PROGRAM valve_manager
VAR
	//Digital valve
	nv_3110_b : valve_digital;
	nv_3210_b : valve_digital;
	nv_3310_b : valve_digital;
	nv_3135_b : valve_digital;
	nv_3235_b : valve_digital;
	nv_3335_b : valve_digital;
	nv_3372_b : valve_digital;
	nv_3162_b : valve_digital;
	
	// Analog Valve Function Block
	av_3148_b : valve_analog;
	av_3248_b : valve_analog;
	av_3348_b : valve_analog;


	//Repeat for each valve?
	u_3112_b_open_request: BOOL;
	u_3112_b_idle_request: BOOL;
	u_3112_b_cip_request: BOOL;
	u_3112_b_manual_request: BOOL;
	u_3112_b_stop_request: BOOL;
	u_3112_b_intlk: BOOL;
	gen_alm_active: BOOL;
	ed_routine_idle: BOOL;
	ed_routine_cip: BOOL;
	ed_routine_manual: BOOL;
	ed_routine_maint: BOOL;
	nv_3110_b_idle_request: BOOL;
	nv_3110_b_cip_request: BOOL;
	nv_3110_b_manual_request: BOOL;
	nv_3110_b_intlk: BOOL;
	nv_3110_b_stop_request: BOOL;
	nv_3110_b_open_request: BOOL;
	nv_3210_b_open_request: BOOL;
	nv_3310_b_open_request: BOOL;
	nv_3135_b_open_request: BOOL;
	nv_3235_b_open_request: BOOL;
	nv_3335_b_open_request: BOOL;
	nv_3372_b_open_request: BOOL;
	nv_3210_b_idle_request: BOOL;
	nv_3210_b_cip_request: BOOL;
	nv_3210_b_manual_request: BOOL;
	nv_3210_b_stop_request: BOOL;
	nv_3210_b_intlk: BOOL;
	
	nv_3310_b_idle_request: BOOL;
	nv_3310_b_cip_request: BOOL;
	nv_3310_b_manual_request: BOOL;
	nv_3310_b_stop_request: BOOL;
	nv_3310_b_intlk: BOOL;
	
	nv_3135_b_idle_request: BOOL;
	nv_3135_b_cip_request: BOOL;
	nv_3135_b_manual_request: BOOL;
	nv_3135_b_stop_request: BOOL;
	nv_3135_b_intlk: BOOL;
	
	nv_3235_b_idle_request: BOOL;
	nv_3235_b_cip_request: BOOL;
	nv_3235_b_manual_request: BOOL;
	nv_3235_b_stop_request: BOOL;
	nv_3235_b_intlk: BOOL;
	
	nv_3335_b_idle_request: BOOL;
	nv_3335_b_cip_request: BOOL;
	nv_3335_b_manual_request: BOOL;
	nv_3335_b_stop_request: BOOL;
	nv_3335_b_intlk: BOOL;
	
	nv_3372_b_idle_request: BOOL;
	nv_3372_b_cip_request: BOOL;
	nv_3372_b_manual_request: BOOL;
	nv_3372_b_stop_request: BOOL;
	nv_3372_b_intlk: BOOL;
	
	nv_3162_b_idle_request: BOOL;
	nv_3162_b_cip_request: BOOL;
	nv_3162_b_manual_request: BOOL;
	nv_3162_b_stop_request: BOOL;
	nv_3162_b_intlk: BOOL;
	nv_3162_b_open_request: BOOL;
	
	av_3148_b_idle_request: BOOL;
	av_3148_b_cip_request: BOOL;
	av_3148_b_idle_position_request: REAL;
	av_3148_b_position_request: REAL;
	av_3148_b_cip_position_request: REAL;
	av_3148_b_manual_position_request: REAL;
	av_3148_b_manual_request: BOOL;
	av_3148_b_maint_request: BOOL;
	av_3148_b_maint_position_request: REAL;
	av_3148_b_intlk: BOOL;
	av_3148_b_stop_request: BOOL;
	av_3148_b_open_request: BOOL;
	
	av_3248_b_idle_request: BOOL;
	av_3248_b_cip_request: BOOL;
	av_3248_b_idle_position_request: REAL;
	av_3248_b_position_request: REAL;
	av_3248_b_cip_position_request: REAL;
	av_3248_b_manual_position_request: REAL;
	av_3248_b_manual_request: BOOL;
	av_3248_b_maint_request: BOOL;
	av_3248_b_maint_position_request: REAL;
	av_3248_b_intlk: BOOL;
	av_3248_b_stop_request: BOOL;
	av_3248_b_open_request: BOOL;
	
	av_3348_b_idle_request: BOOL;
	av_3348_b_cip_request: BOOL;
	av_3348_b_idle_position_request: REAL;
	av_3348_b_position_request: REAL;
	av_3348_b_cip_position_request: REAL;
	av_3348_b_manual_position_request: REAL;
	av_3348_b_manual_request: BOOL;
	av_3348_b_maint_request: BOOL;
	av_3348_b_maint_position_request: REAL;
	av_3348_b_intlk: BOOL;
	av_3348_b_stop_request: BOOL;
	av_3348_b_open_request: BOOL;
	
END_VAR
VAR // added by the converter: edge detectors and wires of the graphical bodies
    _w1, _w2, _w3, _w4, _w5, _w6, _w7, _w8, _w9, _w10, _w11, _w12, _w13, _w14, _w15 : BOOL;
END_VAR

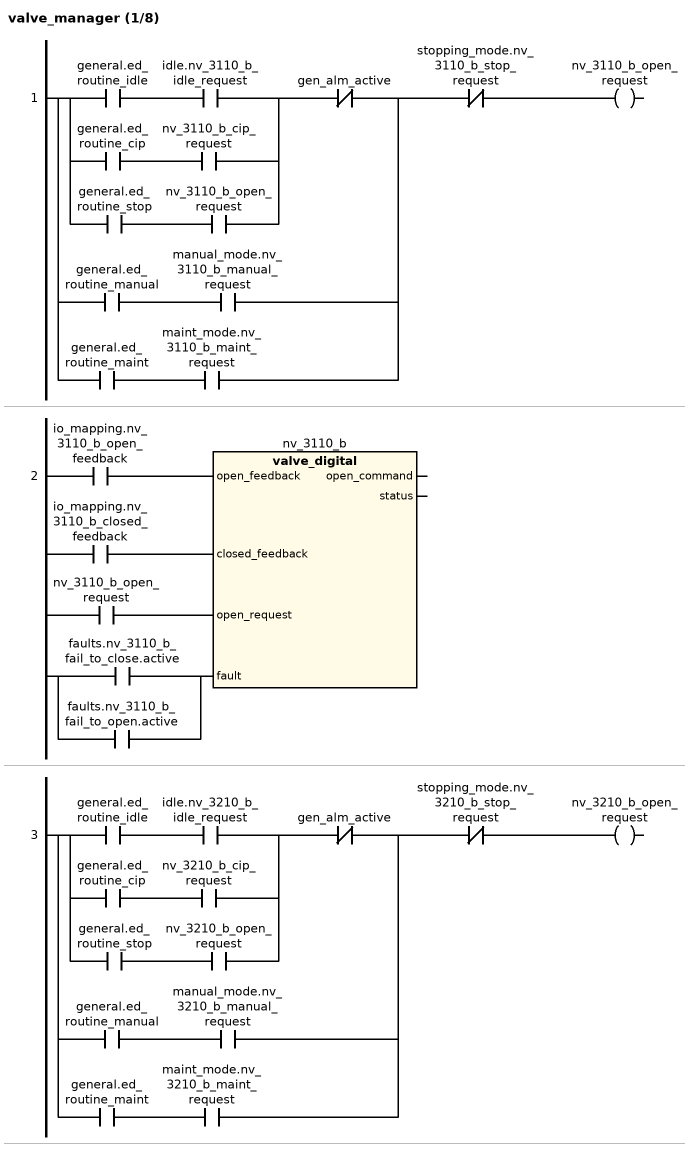
// NETWORK 1
nv_3110_b_open_request := ((general.ed_routine_idle AND idle.nv_3110_b_idle_request OR general.ed_routine_cip AND nv_3110_b_cip_request OR general.ed_routine_stop AND nv_3110_b_open_request) AND NOT gen_alm_active OR general.ed_routine_manual AND manual_mode.nv_3110_b_manual_request OR general.ed_routine_maint AND maint_mode.nv_3110_b_maint_request) AND NOT stopping_mode.nv_3110_b_stop_request;

// NETWORK 2
nv_3110_b(
    open_feedback := io_mapping.nv_3110_b_open_feedback,
    closed_feedback := io_mapping.nv_3110_b_closed_feedback,
    open_request := nv_3110_b_open_request,
    fault := faults.nv_3110_b_fail_to_close.active OR faults.nv_3110_b_fail_to_open.active); // valve_digital

// NETWORK 3
nv_3210_b_open_request := ((general.ed_routine_idle AND idle.nv_3210_b_idle_request OR general.ed_routine_cip AND nv_3210_b_cip_request OR general.ed_routine_stop AND nv_3210_b_open_request) AND NOT gen_alm_active OR general.ed_routine_manual AND manual_mode.nv_3210_b_manual_request OR general.ed_routine_maint AND maint_mode.nv_3210_b_maint_request) AND NOT stopping_mode.nv_3210_b_stop_request;

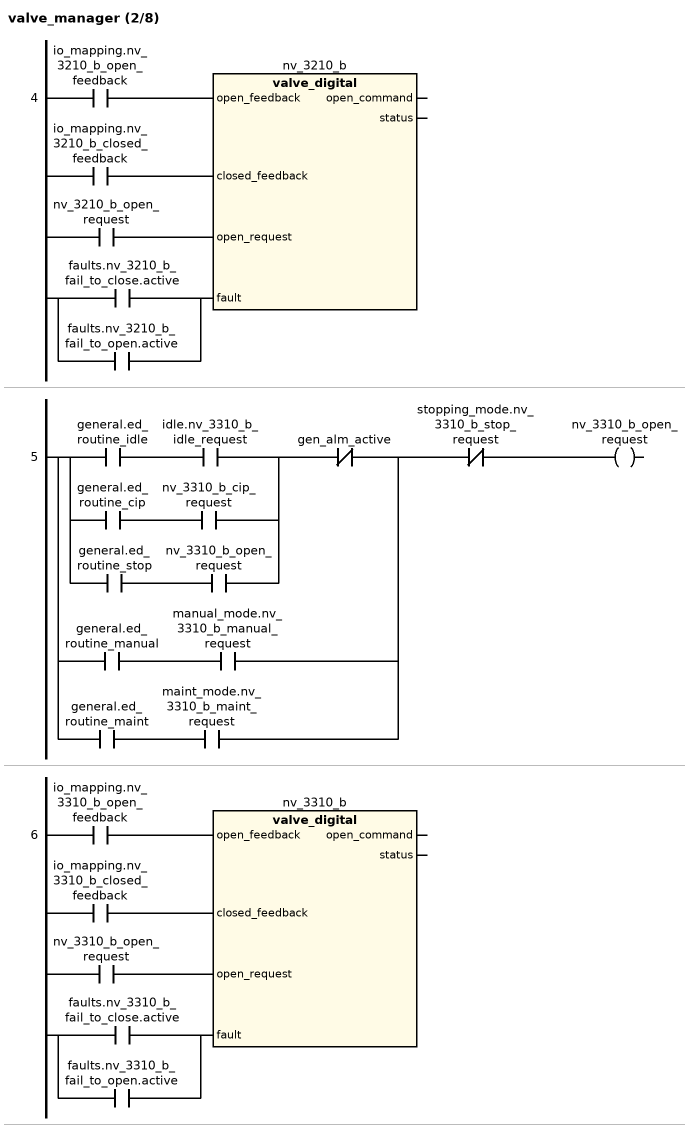
// NETWORK 4
nv_3210_b(
    open_feedback := io_mapping.nv_3210_b_open_feedback,
    closed_feedback := io_mapping.nv_3210_b_closed_feedback,
    open_request := nv_3210_b_open_request,
    fault := faults.nv_3210_b_fail_to_close.active OR faults.nv_3210_b_fail_to_open.active); // valve_digital

// NETWORK 5
nv_3310_b_open_request := ((general.ed_routine_idle AND idle.nv_3310_b_idle_request OR general.ed_routine_cip AND nv_3310_b_cip_request OR general.ed_routine_stop AND nv_3310_b_open_request) AND NOT gen_alm_active OR general.ed_routine_manual AND manual_mode.nv_3310_b_manual_request OR general.ed_routine_maint AND maint_mode.nv_3310_b_maint_request) AND NOT stopping_mode.nv_3310_b_stop_request;

// NETWORK 6
nv_3310_b(
    open_feedback := io_mapping.nv_3310_b_open_feedback,
    closed_feedback := io_mapping.nv_3310_b_closed_feedback,
    open_request := nv_3310_b_open_request,
    fault := faults.nv_3310_b_fail_to_close.active OR faults.nv_3310_b_fail_to_open.active); // valve_digital

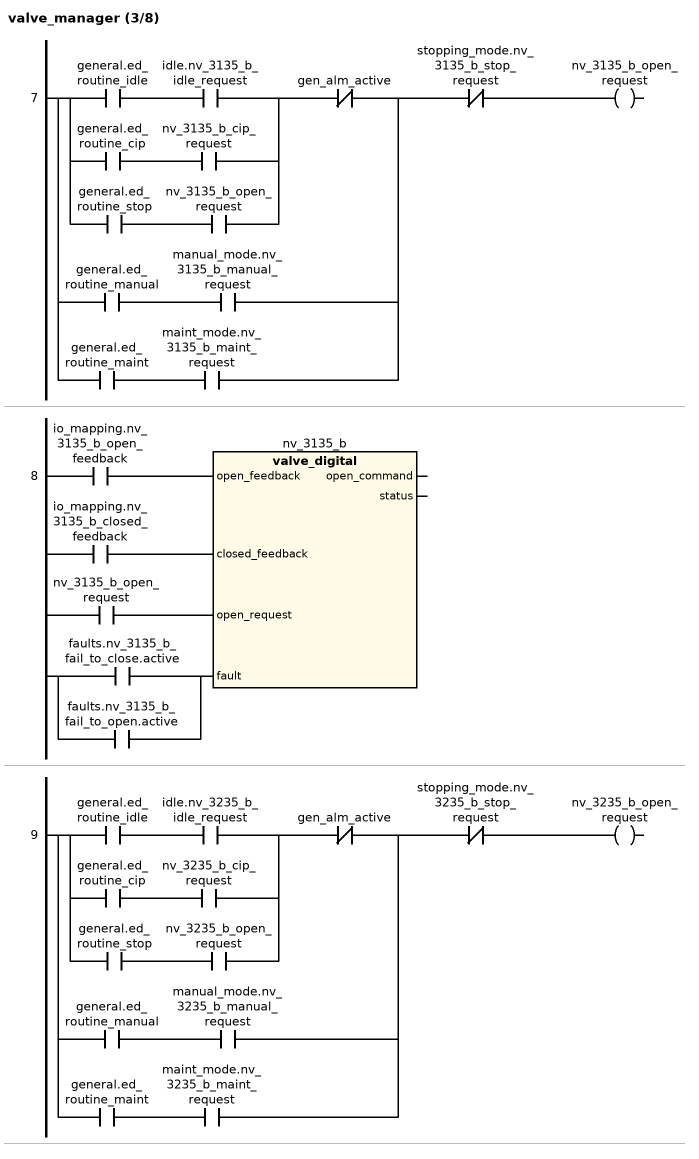
// NETWORK 7
nv_3135_b_open_request := ((general.ed_routine_idle AND idle.nv_3135_b_idle_request OR general.ed_routine_cip AND nv_3135_b_cip_request OR general.ed_routine_stop AND nv_3135_b_open_request) AND NOT gen_alm_active OR general.ed_routine_manual AND manual_mode.nv_3135_b_manual_request OR general.ed_routine_maint AND maint_mode.nv_3135_b_maint_request) AND NOT stopping_mode.nv_3135_b_stop_request;

// NETWORK 8
nv_3135_b(
    open_feedback := io_mapping.nv_3135_b_open_feedback,
    closed_feedback := io_mapping.nv_3135_b_closed_feedback,
    open_request := nv_3135_b_open_request,
    fault := faults.nv_3135_b_fail_to_close.active OR faults.nv_3135_b_fail_to_open.active); // valve_digital

// NETWORK 9
nv_3235_b_open_request := ((general.ed_routine_idle AND idle.nv_3235_b_idle_request OR general.ed_routine_cip AND nv_3235_b_cip_request OR general.ed_routine_stop AND nv_3235_b_open_request) AND NOT gen_alm_active OR general.ed_routine_manual AND manual_mode.nv_3235_b_manual_request OR general.ed_routine_maint AND maint_mode.nv_3235_b_maint_request) AND NOT stopping_mode.nv_3235_b_stop_request;

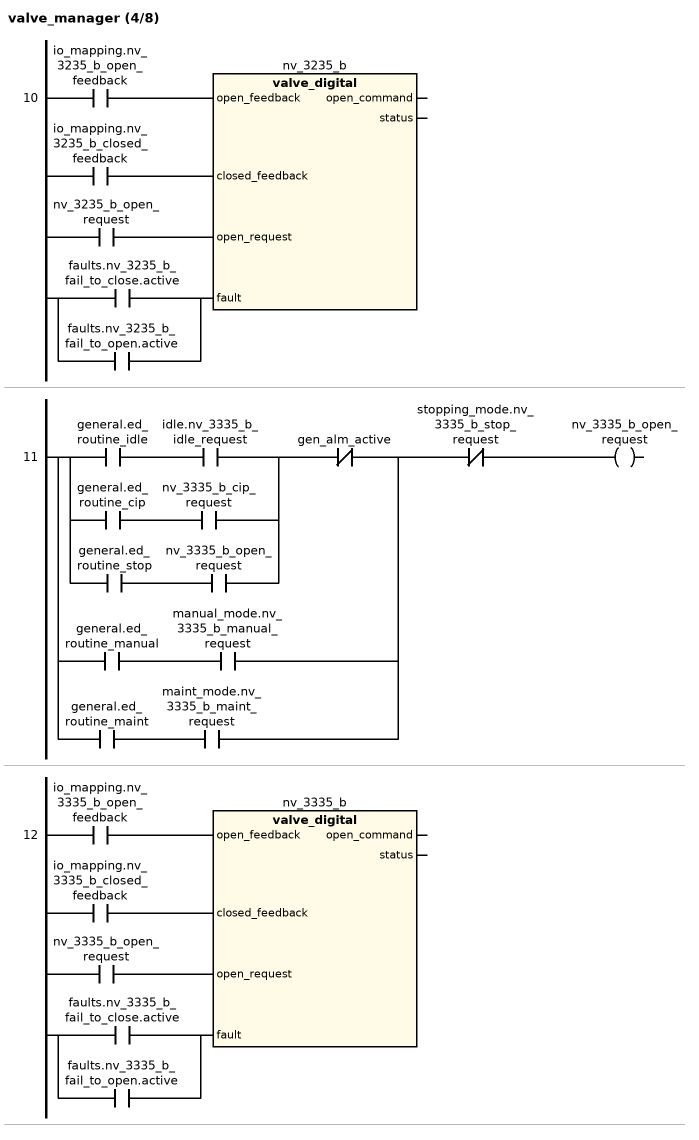
// NETWORK 10
nv_3235_b(
    open_feedback := io_mapping.nv_3235_b_open_feedback,
    closed_feedback := io_mapping.nv_3235_b_closed_feedback,
    open_request := nv_3235_b_open_request,
    fault := faults.nv_3235_b_fail_to_close.active OR faults.nv_3235_b_fail_to_open.active); // valve_digital

// NETWORK 11
nv_3335_b_open_request := ((general.ed_routine_idle AND idle.nv_3335_b_idle_request OR general.ed_routine_cip AND nv_3335_b_cip_request OR general.ed_routine_stop AND nv_3335_b_open_request) AND NOT gen_alm_active OR general.ed_routine_manual AND manual_mode.nv_3335_b_manual_request OR general.ed_routine_maint AND maint_mode.nv_3335_b_maint_request) AND NOT stopping_mode.nv_3335_b_stop_request;

// NETWORK 12
nv_3335_b(
    open_feedback := io_mapping.nv_3335_b_open_feedback,
    closed_feedback := io_mapping.nv_3335_b_closed_feedback,
    open_request := nv_3335_b_open_request,
    fault := faults.nv_3335_b_fail_to_close.active OR faults.nv_3335_b_fail_to_open.active); // valve_digital

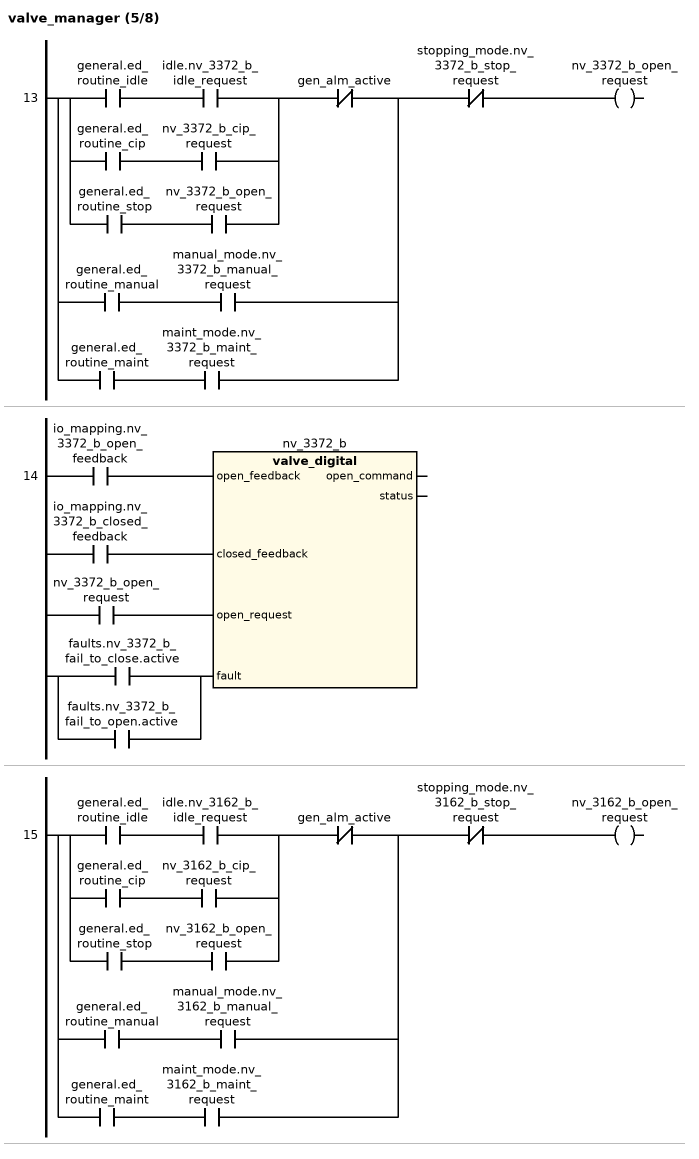
// NETWORK 13
nv_3372_b_open_request := ((general.ed_routine_idle AND idle.nv_3372_b_idle_request OR general.ed_routine_cip AND nv_3372_b_cip_request OR general.ed_routine_stop AND nv_3372_b_open_request) AND NOT gen_alm_active OR general.ed_routine_manual AND manual_mode.nv_3372_b_manual_request OR general.ed_routine_maint AND maint_mode.nv_3372_b_maint_request) AND NOT stopping_mode.nv_3372_b_stop_request;

// NETWORK 14
nv_3372_b(
    open_feedback := io_mapping.nv_3372_b_open_feedback,
    closed_feedback := io_mapping.nv_3372_b_closed_feedback,
    open_request := nv_3372_b_open_request,
    fault := faults.nv_3372_b_fail_to_close.active OR faults.nv_3372_b_fail_to_open.active); // valve_digital

// NETWORK 15
nv_3162_b_open_request := ((general.ed_routine_idle AND idle.nv_3162_b_idle_request OR general.ed_routine_cip AND nv_3162_b_cip_request OR general.ed_routine_stop AND nv_3162_b_open_request) AND NOT gen_alm_active OR general.ed_routine_manual AND manual_mode.nv_3162_b_manual_request OR general.ed_routine_maint AND maint_mode.nv_3162_b_maint_request) AND NOT stopping_mode.nv_3162_b_stop_request;

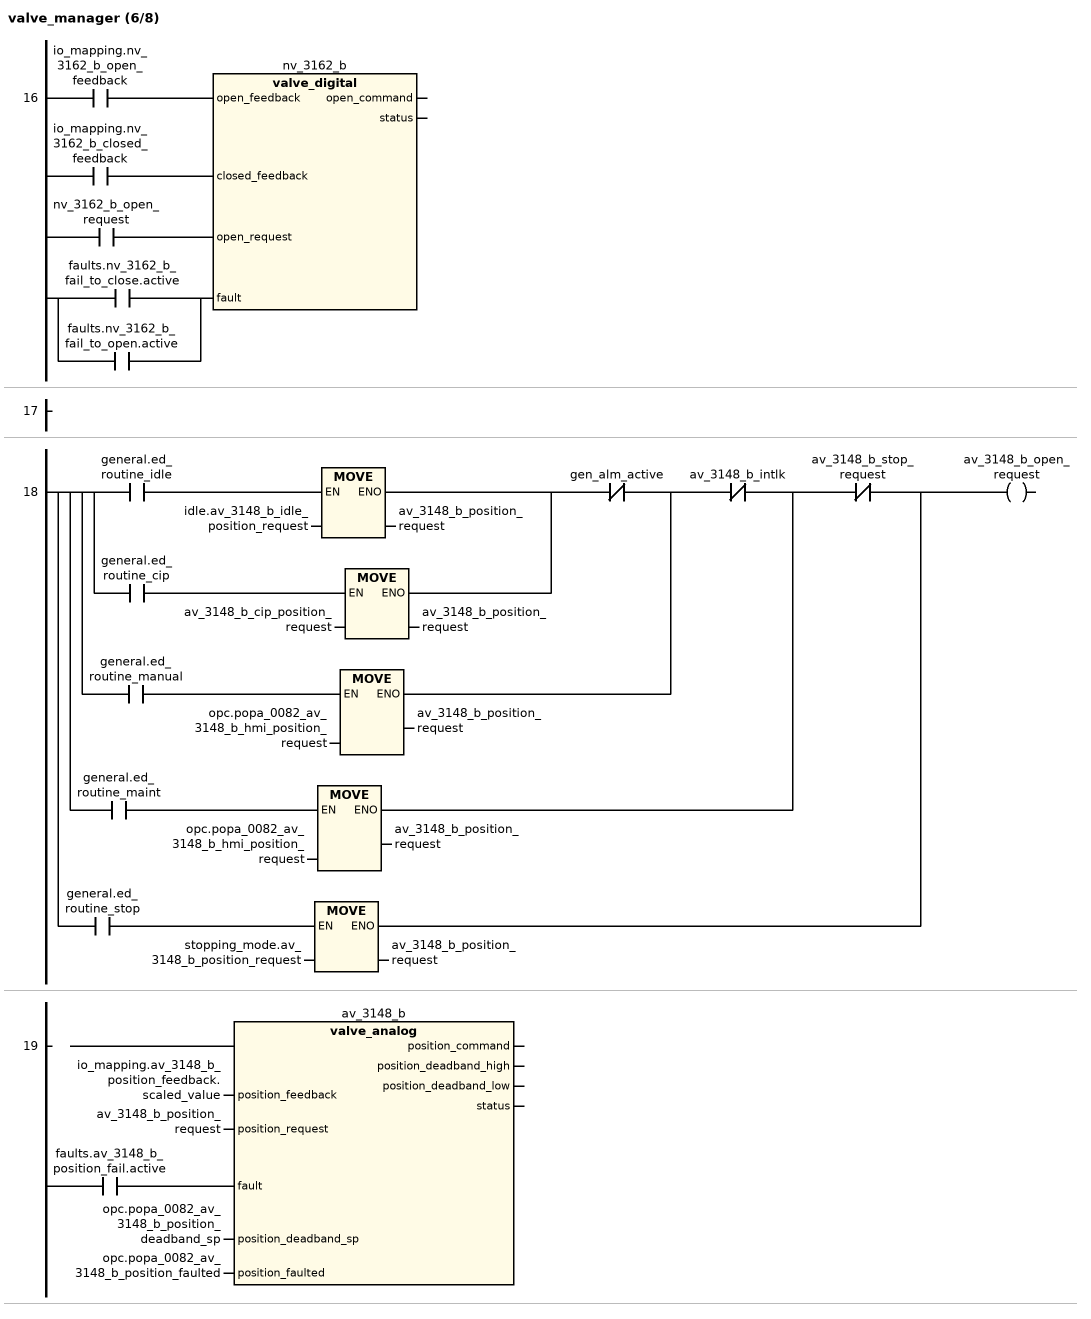
// NETWORK 16
nv_3162_b(
    open_feedback := io_mapping.nv_3162_b_open_feedback,
    closed_feedback := io_mapping.nv_3162_b_closed_feedback,
    open_request := nv_3162_b_open_request,
    fault := faults.nv_3162_b_fail_to_close.active OR faults.nv_3162_b_fail_to_open.active); // valve_digital

// NETWORK 17

// NETWORK 18
_w1 := general.ed_routine_idle;
IF _w1 THEN av_3148_b_position_request := idle.av_3148_b_idle_position_request; END_IF
_w2 := general.ed_routine_cip;
IF _w2 THEN av_3148_b_position_request := av_3148_b_cip_position_request; END_IF
_w3 := general.ed_routine_manual;
IF _w3 THEN av_3148_b_position_request := opc.popa_0082_av_3148_b_hmi_position_request; END_IF
_w4 := general.ed_routine_maint;
IF _w4 THEN av_3148_b_position_request := opc.popa_0082_av_3148_b_hmi_position_request; END_IF
_w5 := general.ed_routine_stop;
IF _w5 THEN av_3148_b_position_request := stopping_mode.av_3148_b_position_request; END_IF
av_3148_b_open_request := (((_w1 OR _w2) AND NOT gen_alm_active OR _w3) AND NOT av_3148_b_intlk OR _w4) AND NOT av_3148_b_stop_request OR _w5;

// NETWORK 19
av_3148_b(
    position_feedback := io_mapping.av_3148_b_position_feedback.scaled_value,
    position_request := av_3148_b_position_request,
    fault := faults.av_3148_b_position_fail.active,
    position_deadband_sp := opc.popa_0082_av_3148_b_position_deadband_sp,
    position_faulted := opc.popa_0082_av_3148_b_position_faulted); // valve_analog

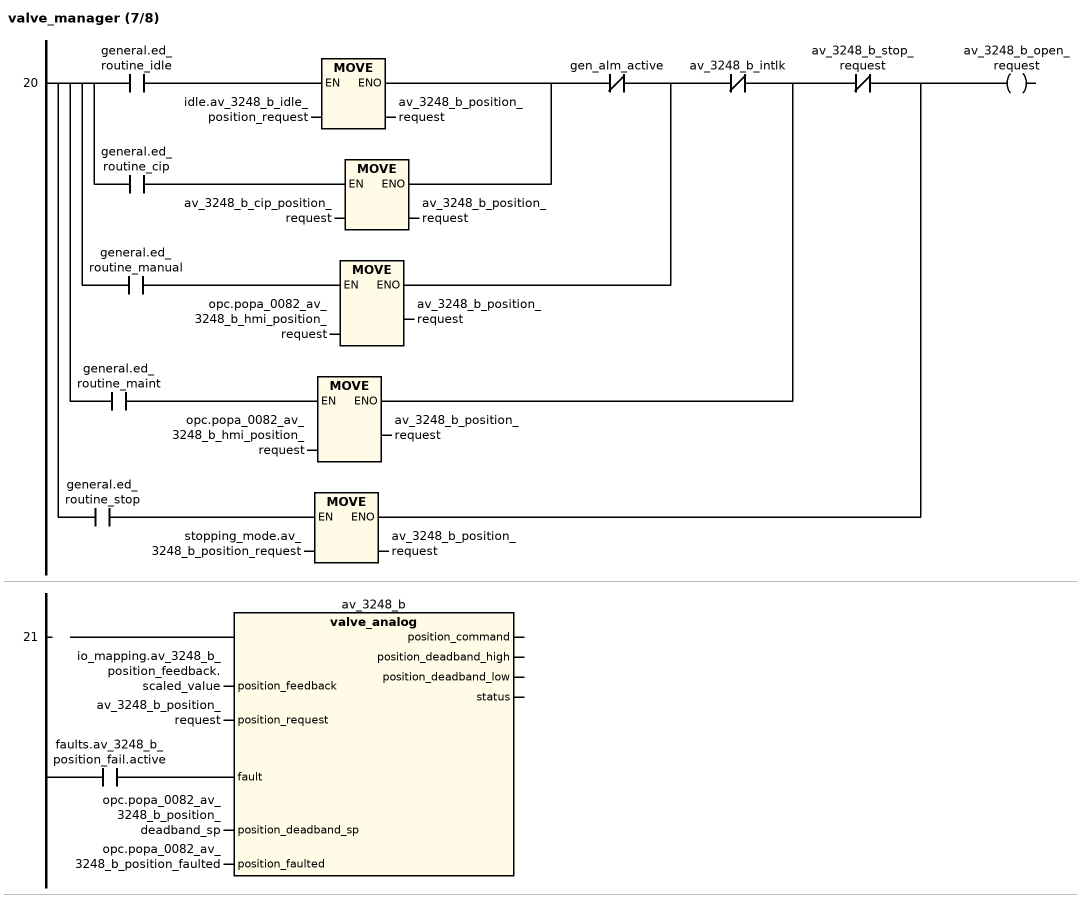
// NETWORK 20
_w6 := general.ed_routine_idle;
IF _w6 THEN av_3248_b_position_request := idle.av_3248_b_idle_position_request; END_IF
_w7 := general.ed_routine_cip;
IF _w7 THEN av_3248_b_position_request := av_3248_b_cip_position_request; END_IF
_w8 := general.ed_routine_manual;
IF _w8 THEN av_3248_b_position_request := opc.popa_0082_av_3248_b_hmi_position_request; END_IF
_w9 := general.ed_routine_maint;
IF _w9 THEN av_3248_b_position_request := opc.popa_0082_av_3248_b_hmi_position_request; END_IF
_w10 := general.ed_routine_stop;
IF _w10 THEN av_3248_b_position_request := stopping_mode.av_3248_b_position_request; END_IF
av_3248_b_open_request := (((_w6 OR _w7) AND NOT gen_alm_active OR _w8) AND NOT av_3248_b_intlk OR _w9) AND NOT av_3248_b_stop_request OR _w10;

// NETWORK 21
av_3248_b(
    position_feedback := io_mapping.av_3248_b_position_feedback.scaled_value,
    position_request := av_3248_b_position_request,
    fault := faults.av_3248_b_position_fail.active,
    position_deadband_sp := opc.popa_0082_av_3248_b_position_deadband_sp,
    position_faulted := opc.popa_0082_av_3248_b_position_faulted); // valve_analog

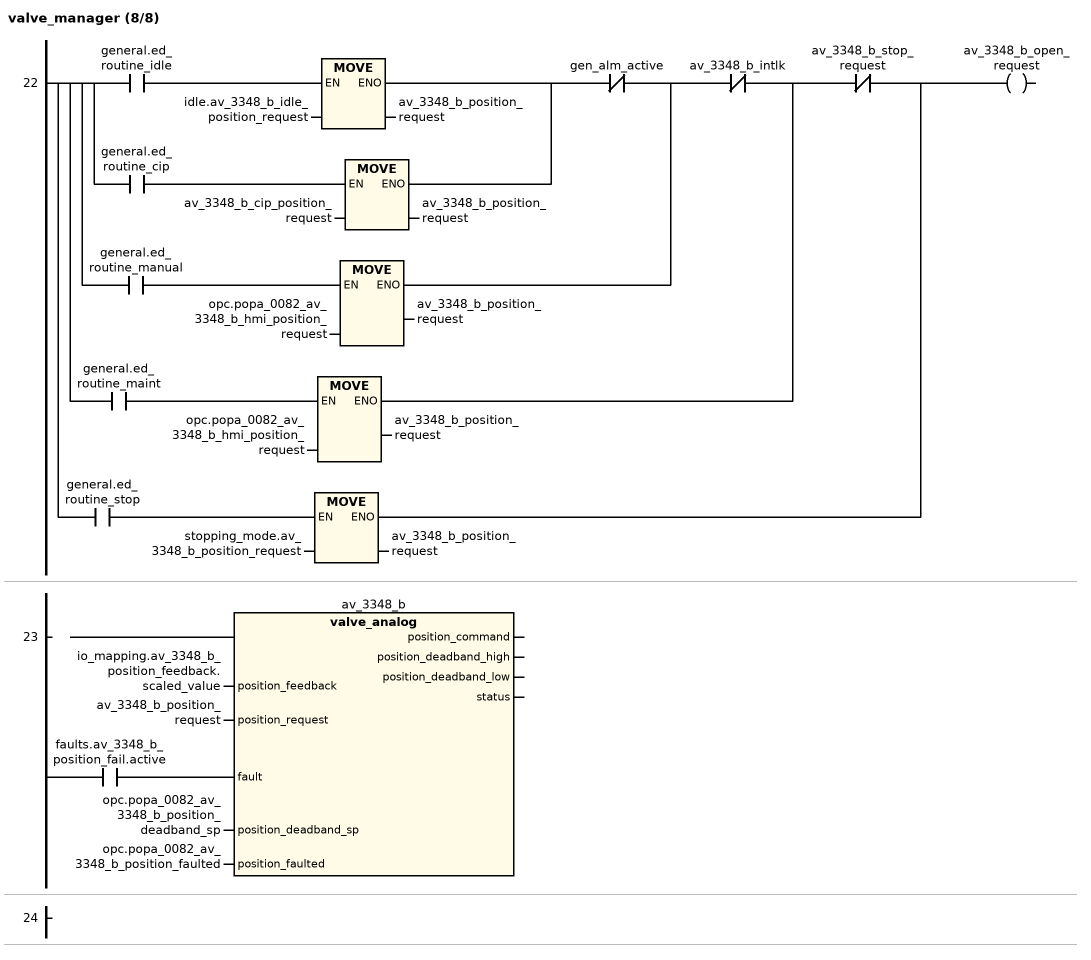
// NETWORK 22
_w11 := general.ed_routine_idle;
IF _w11 THEN av_3348_b_position_request := idle.av_3348_b_idle_position_request; END_IF
_w12 := general.ed_routine_cip;
IF _w12 THEN av_3348_b_position_request := av_3348_b_cip_position_request; END_IF
_w13 := general.ed_routine_manual;
IF _w13 THEN av_3348_b_position_request := opc.popa_0082_av_3348_b_hmi_position_request; END_IF
_w14 := general.ed_routine_maint;
IF _w14 THEN av_3348_b_position_request := opc.popa_0082_av_3348_b_hmi_position_request; END_IF
_w15 := general.ed_routine_stop;
IF _w15 THEN av_3348_b_position_request := stopping_mode.av_3348_b_position_request; END_IF
av_3348_b_open_request := (((_w11 OR _w12) AND NOT gen_alm_active OR _w13) AND NOT av_3348_b_intlk OR _w14) AND NOT av_3348_b_stop_request OR _w15;

// NETWORK 23
av_3348_b(
    position_feedback := io_mapping.av_3348_b_position_feedback.scaled_value,
    position_request := av_3348_b_position_request,
    fault := faults.av_3348_b_position_fail.active,
    position_deadband_sp := opc.popa_0082_av_3348_b_position_deadband_sp,
    position_faulted := opc.popa_0082_av_3348_b_position_faulted); // valve_analog

// NETWORK 24

END_PROGRAM

(* stored: Version 1.1.0.1, ProductVersion 3.1.4024.15
   POU valve_manager: Id {359c8254-c75f-419b-be16-97d4ba9197db}, SpecialFunc None *)
